PROGRAM Greiferansteuerung
VAR
	greiferSignal AT%I*:LREAL:=0;
	greiferEnable AT%Q*:BOOL:=0;
	greiferValue  AT%Q* :INT:=0;
	
	greiferSliderFromIO 	AT%I*:BOOL:=0;
	greiferSliderToSimulink AT%Q*:LREAL:=0;
	
	greiferLichtschrankeFromIO AT%I*:BOOL:=0;
	greiferLichtschrankeToSimulink AT%Q*:LREAL:=0;
END_VAR

IF greiferSignal=0 THEN
	greiferEnable:=1;
	greiferValue:=-32767;
ELSE
	greiferEnable:=1;
	greiferValue:=32767;
END_IF

greiferSliderToSimulink:=BOOL_TO_LREAL(NOT(greiferSliderFromIO));
greiferLichtschrankeToSimulink:=BOOL_TO_LREAL(NOT(greiferLichtschrankeFromIO));

END_PROGRAM

(* stored: Version 1.1.0.1, ProductVersion 3.1.4022.3
   POU Greiferansteuerung: Id {914b4c40-8d67-4edc-a810-6f17709861da}, SpecialFunc None *)
